PROGRAM PLC_PRG
VAR

END_VAR

PRG_Cell();

RETURN;

END_PROGRAM

(* stored: Version 1.1.0.1, ProductVersion 3.1.4024.9
   POU PLC_PRG: Id {cf366734-d49e-4bbc-8306-bebddd2306df}, SpecialFunc None *)
